TYPE ENUM_SLOT :
(
	SLOT_1 := 1,
	SLOT_2,
	SLOT_3,
	SLOT_4,
	SLOT_LAST
);
END_TYPE

(* stored: Version 1.1.0.1, ProductVersion 3.1.4024.10
   DUT ENUM_SLOT: Id {08360d0a-85a6-4281-9a08-ab8848cdf16e} *)
